// SIMATIC S7-200 SMART project (STEP 7-Micro/WIN SMART), CPU ST30

SYMBOL_TABLE System Symbols
Always_On        SM0.0    // Always ON
END_SYMBOL_TABLE

ORGANIZATION_BLOCK MAIN:OB1
TITLE=Program Comments
BEGIN
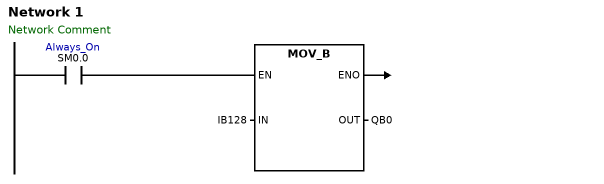
Network 1
// Network Comment
LD     Always_On:SM0.0
MOVB   IB128, QB0
END_ORGANIZATION_BLOCK
